// TwinCAT 3 PLC project train
// ProgramVersion: 3.1.4026.17
// libraries:
//   Tc2_ModbusRTU, * (Beckhoff Automation GmbH)
//   Tc2_SerialCom, * (Beckhoff Automation GmbH)
//   Tc2_Standard, * (Beckhoff Automation GmbH)
//   Tc2_System, * (Beckhoff Automation GmbH)
// project tree:
//   / PlcTask.TcTTO
//   POUs/ FB_Start.TcPOU, MAIN.TcPOU, RIFD.TcPOU, FB_SerialCOM.TcPOU
// real-time tasks:
//   TASK PlcTask: cycle T#2ms, priority 20, ADS port 350
// I/O:
//   DEVICE Gerät 1 (EtherCAT), AmsNetId 10.201.9.16.2.1
//     Klemme 7 (EK1100) [EK1100 EtherCAT-Koppler (2A E-Bus)]
//       Klemme 8 (EL1859) [EL1859 8K. Dig. Eingang 24V, 3ms, 8K. Dig. Ausgang 24V, 0.5A]
//       Klemme 9 (EL1904) [EL1904, 4 K. Safety Eingang 24V, TwinSAFE]
//         modules: Module 1 (FSOES)
//       Klemme 10 (EL3312) [EL3312 2K. Ana. Eingang Thermoelement (TC)]
//       Klemme 11 (EL5021-0090) [EL5021-0090 1K. Sin/Cos Encoder, TwinSAFE SC]
//       Klemme 12 (EL3255) [EL3255 5K. Potentiometerauswertung mit Sensorversorgung]
//       Klemme 13 (EL3214-0090) [EL3214-0090 4K. Ana. Eingang PT100 (RTD), TwinSAFE SC]
//       Klemme 14 (EL6001) [EL6001 Schnittstelle (RS232)]
//       Klemme 15 (EL2502) [EL2502 2K. PWM Ausgang, 24V]
//       Klemme 16 (EL9505) [EL9505 Netzteilklemme 5V]
//       Klemme 22 (EL9011) [EL9011 Endklemme]
//     Klemme 1 (EK1100) [EK1100 EtherCAT-Koppler (2A E-Bus)]
//       Klemme 2 (EL1012) [EL1012 2K. Dig. Eingang 24V, 10µs]
//       Klemme 3 (EL2624) [EL2624 4K. Relais Ausgang, Schließer (125V AC / 30V DC)]
//       Klemme 4 (EL2624) [EL2624 4K. Relais Ausgang, Schließer (125V AC / 30V DC)]
//       Klemme 5 (EL6002) [EL6002 Schnittstelle 2K. (RS232)]
//       Klemme 6 (EL9011) [EL9011 Endklemme]
// variable links:
//   train/train Instance <-> Device 1 (EtherCAT)/Term 1 (EK1100)/Term 3 (EL2624)
//     PlcTask Outputs/RIFD.bGleis{1..4} <-> Channel {1..4}/Output  (4 links)
//   train/train Instance <-> Device 1 (EtherCAT)/Term 1 (EK1100)/Term 4 (EL2624)
//     PlcTask Outputs/RIFD.fbStart.bLamp <-> Channel 2/Output
//   train/train Instance <-> Device 1 (EtherCAT)/Term 1 (EK1100)/Term 5 (EL6002)
//     PlcTask Inputs/RIFD.fbSerCom.EL6InData/D <-> COM Inputs Channel 1/Data In 0
//     PlcTask Inputs/RIFD.fbSerCom.EL6InData/D @bit {8..168 step 8} <-> COM Inputs Channel 1/Data In {1..21}  (21 links)
//     PlcTask Inputs/RIFD.fbSerCom.EL6InData/Status <-> COM Inputs Channel 1/Status
//     PlcTask Outputs/RIFD.fbSerCom.EL6OutData/Ctrl <-> COM Outputs Channel 1/Ctrl
//     PlcTask Outputs/RIFD.fbSerCom.EL6OutData/D <-> COM Outputs Channel 1/Data Out 0
//     PlcTask Outputs/RIFD.fbSerCom.EL6OutData/D @bit {8..168 step 8} <-> COM Outputs Channel 1/Data Out {1..21}  (21 links)
//   train/train Instance <-> Device 1 (EtherCAT)/Term 7 (EK1100)/Term 8 (EL1859)
//     PlcTask Inputs/RIFD.fbStart.bSwitch <-> Channel 1/Input
//     PlcTask Outputs/RIFD.fbStart.bLamp <-> Channel 9/Output

CONFIGURATION train
    RESOURCE PLC ON TwinCAT3
        TASK PlcTask(INTERVAL := T#2ms, PRIORITY := 20);
        PROGRAM MAIN WITH PlcTask : MAIN;
    END_RESOURCE
END_CONFIGURATION

// ---- POUs/MAIN.TcPOU
PROGRAM MAIN
VAR
END_VAR


RIFD();

END_PROGRAM

// ---- POUs/RIFD.TcPOU
PROGRAM RIFD
VAR
	//bSensor AT%I* : BOOL;
	bGleis1 AT%Q* : BOOL;
	bGleis2 AT%Q* : BOOL;
	
	bGleis3 AT%Q* : BOOL;
	bGleis4 AT%Q* : BOOL;
	
	//bSenor: BOOL;
	
	fbTonWeiche : TON;
	
	fbSerCom	: FB_SerialCom; 
	nTransponderOld : INT;
	
	fbStart : FB_Start;
END_VAR


fbStart();

fbSerCom(nTransponderID=> );



//bGleis1 := bSenor; 
//IF bSensor = TRUE THEN
	///bGleis1 := TRUE;
	
//END_IF

IF NOT (fbSerCom.nTransponderID = nTransponderOld) THEN
	CASE fbSerCom.nTransponderID OF
		0:
			;
		1:
			bGleis2 := TRUE;
			fbTonWeiche.IN := TRUE;
			nTransponderOld := fbSerCom.nTransponderID ;
			
		7:
			bGleis1 := TRUE;
			fbTonWeiche.IN := TRUE;
			nTransponderOld := fbSerCom.nTransponderID ;
			
		255:
			bGleis2 := TRUE;
			bGleis3 := TRUE;
			fbTonWeiche.IN := TRUE;
			nTransponderOld := fbSerCom.nTransponderID ;
				
		8:
			bGleis2 := TRUE;
			bGleis4 := TRUE;
			fbTonWeiche.IN := TRUE;
			nTransponderOld := fbSerCom.nTransponderID ;
		ELSE
			;
			
	END_CASE
ELSE
	;
END_IF


// Weichenstrom abschalten

fbTonWeiche(IN:=  , PT:= T#250MS , Q=> , ET=> );
IF fbTonWeiche.Q  THEN
 bGleis1 := bGleis2:= bGleis3 := bGleis4 := FALSE;
 fbTonWeiche.IN := FALSE;
END_IF

END_PROGRAM

// ---- POUs/FB_SerialCOM.TcPOU
// CoE-Settings EL6002
// 0x8000:05 : TRUE
// 0x8000:11 : 9600
// 0x8000:15 : 8E1(4)

FUNCTION_BLOCK FB_SerialCOM
VAR_INPUT
END_VAR
VAR_OUTPUT
		nTransponderID	: INT; // latest Transponder ID
END_VAR
VAR
	//  instances
	fbSerLineControl				: SerialLineControl;
	fbRcvData						: ReceiveData;
	// data structures
	stComBufferIn, stComBufferOut	: ComBuffer;
	EL6InData AT%I*					: EL6inData22B;
	EL6OutData AT%Q*				: EL6outData22B;

	// ReceiveData
	nPrefix		: BYTE := 2; // fixed defined prefix char
	nSuffix		: BYTE := 0; // no suffix char
	nRecvData	: ARRAY[1..4] OF BYTE; // contains prefix, data and crc

	
END_VAR

// SerialLine DataControl
fbSerLineControl(
	Mode:= Seriallinemode_EL6_22B, 
	pComIn:= ADR(EL6InData), 
	pComOut:= ADR(EL6OutData), 
	SizeComIn:= SIZEOF(EL6InData), 
	Error=> , 
	ErrorID=> , 
	TxBuffer:= stComBufferOut, 
	RxBuffer:= stComBufferIn
	);

// Receive Data Transponder
// Prefis := 02
// Length Prefix := 1 Byte
// Data = 2 Byte
// CRC = 1 Byte

// data receiver	
fbRcvData(
	pPrefix:= ADR(nPrefix), 
	LenPrefix:= 1, // length prefix = 1 Byte
	pSuffix:= ADR(nSuffix), 
	LenSuffix:= 0,  // no suffix char available
	pReceiveData:= ADR(nRecvData), // data array for received data 
	SizeReceiveData:= SIZEOF(nRecvData), 
	Timeout:= T#3S, 
	Reset:= , 
	DataReceived=> , 
	busy=> , 
	Error=> , 
	RxTimeout=> , 
	LenReceiveData=> , 
	RXbuffer:= stComBufferIn);

nTransponderID := BYTE_TO_INT(nRecvData[3]); // extract latest Transponder ID from Serial Port

END_FUNCTION_BLOCK

// ---- POUs/FB_Start.TcPOU
FUNCTION_BLOCK FB_Start
VAR_INPUT
END_VAR
VAR_OUTPUT
END_VAR
VAR
	bSwitch AT%I* : BOOL; 
	bLamp   AT%Q* : BOOL; 
nCaseIndex : INT;
	nGleis: BOOL;
END_VAR


bLamp := bSwitch;
CASE nCaseIndex OF 
0: 	
	IF bSwitch = TRUE  THEN
		nCaseIndex := 10; 
	END_IF;; 
	
10: 
	

	IF bSwitch = TRUE  THEN
		nGleis := TRUE;
	
	ELSE
		nGleis := FALSE;
	END_IF;; 
	
END_CASE

END_FUNCTION_BLOCK
